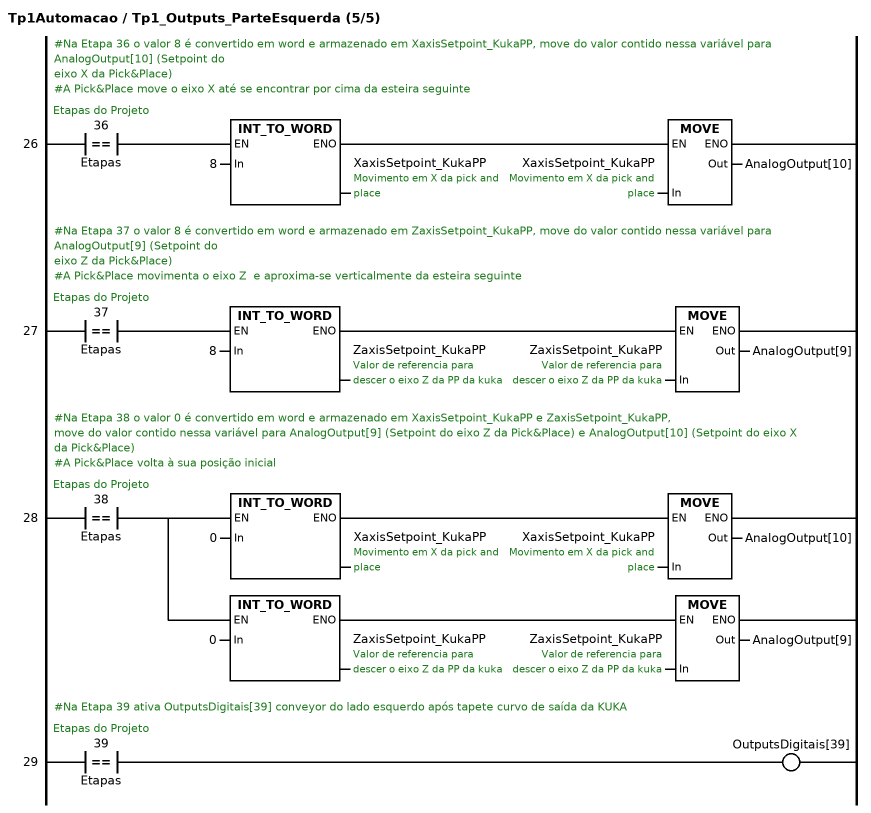
(* [picture p24: Tp1Automacao / Tp1_Outputs_ParteEsquerda, rungs 26-29] *)
(* Rung 26: #Na Etapa 36 o valor 8 é convertido em word e armazenado em XaxisSetpoint_KukaPP, move do valor contido nessa variável para AnalogOutput[10] (Setpoint do / eixo X da Pick&Place) / #A Pick&Place move o eixo X até se encontrar por cima da esteira seguinte *)
IF 36 = Etapas THEN
    XaxisSetpoint_KukaPP := INT_TO_WORD(In := 8);
    AnalogOutput[10] := XaxisSetpoint_KukaPP;
END_IF;
(* Rung 27: #Na Etapa 37 o valor 8 é convertido em word e armazenado em ZaxisSetpoint_KukaPP, move do valor contido nessa variável para AnalogOutput[9] (Setpoint do / eixo Z da Pick&Place) / #A Pick&Place movimenta o eixo Z  e aproxima-se verticalmente da esteira seguinte *)
IF 37 = Etapas THEN
    ZaxisSetpoint_KukaPP := INT_TO_WORD(In := 8);
    AnalogOutput[9] := ZaxisSetpoint_KukaPP;
END_IF;
(* Rung 28: #Na Etapa 38 o valor 0 é convertido em word e armazenado em XaxisSetpoint_KukaPP e ZaxisSetpoint_KukaPP, / move do valor contido nessa variável para AnalogOutput[9] (Setpoint do eixo Z da Pick&Place) e AnalogOutput[10] (Setpoint do eixo X da Pick&Place) / #A Pick&Place volta à sua posição inicial *)
IF 38 = Etapas THEN
    XaxisSetpoint_KukaPP := INT_TO_WORD(In := 0);
    AnalogOutput[10] := XaxisSetpoint_KukaPP;
    ZaxisSetpoint_KukaPP := INT_TO_WORD(In := 0);
    AnalogOutput[9] := ZaxisSetpoint_KukaPP;
END_IF;
(* Rung 29: #Na Etapa 39 ativa OutputsDigitais[39] conveyor do lado esquerdo após tapete curvo de saída da KUKA *)
OutputsDigitais[39] := 39 = Etapas;
END_PROGRAM